# EPICS alarm handler configuration: mps_database/bareTest/alarms/areas/mpln_sph_mp06.alhConfig
GROUP NULL MPLN:SPH:MP06:1
$ALIAS MPS Link Node 125
$GUIDANCE
LTUH MPS
   Group Name: MPLN:SPH:MP06:1
   Summary PV:  MPLN:SPH:MP06:1:STATSUMY
$END
CHANNEL  MPLN:SPH:MP06:1    MPLN:SPH:MP06:1:MPS_EN_RBV		-----
CHANNEL  MPLN:SPH:MP06:1    MPLN:SPH:MP06:1:LC1_MODE_RBV		-----
